PROGRAM DataLogic
VAR	

END_VAR

CASE GVL_Global.data2rcv.cmd[0] OF 
	0: 
		GVL_Global.ModWrite.System_state_control:=2;	// Stop command
	1:
		GVL_Global.ModWrite.System_state_control := 6; // RUN command 
		//battry on, 
		
END_CASE

CASE GVL_Global.data2rcv.cmd[1] OF
	0: 
		GVL_Global.ModWrite.System_mode_control := 2; // Disconnected 
	1:
		GVL_Global.ModWrite.System_mode_control := 3; //Connected	
	2:
		GVL_Global.ModWrite.System_mode_control := 1; // Operational	
		
END_CASE

END_PROGRAM

(* stored: Version 1.1.0.1, ProductVersion 3.1.4024.11
   POU DataLogic: Id {085bc544-972e-46c8-8d94-cedf826394e0}, SpecialFunc None *)
